// TIA Portal V21 export
DATA_BLOCK "AoDb"   // DB106
// stored: AutoNumber false, InstanceOfName AoFb, InstanceOfType FB
"AoFb"
   // VAR_INPUT
   //    AlwaysTrue : Bool;
   //    AlwaysFalse : Bool;
   // END_VAR
   // VAR
   //    Ao01 { S7_SetPoint := 'True'} : "AnalogOutputScaling";   // Mm01Ref
   //    Ao02 { S7_SetPoint := 'True'} : "AnalogOutputScaling";   // Cp01Ref
   //    Ao03 { S7_SetPoint := 'True'} : "AnalogOutputScaling";   // Cv01
   //    Ao04 { S7_SetPoint := 'True'} : "AnalogOutputScaling";   // AoSpare1
   //    Ao05 { S7_SetPoint := 'True'} : "AnalogOutputScaling";   // AoSpare2
   //    Ao06 { S7_SetPoint := 'True'} : "AnalogOutputScaling";   // AoSpare3
   //    Ao07 { S7_SetPoint := 'True'} : "AnalogOutputScaling";   // AoSpare4
   //    Ao08 { S7_SetPoint := 'True'} : "AnalogOutputScaling";   // AoSpare5
   // END_VAR
BEGIN
   Ao01.MinOperatingRpm := 50.0;
   Ao01.MaxOperatingRpm := 400.0;
   Ao01.MaxRpm := 400.0;
   Ao02.MinOperatingRpm := 800.0;
   Ao02.MaxOperatingRpm := 2880.0;
   Ao02.MaxRpm := 2880.0;
   Ao03.MaxOperatingRpm := 100.0;
   Ao03.MaxRpm := 100.0;
END_DATA_BLOCK
